{attribute 'linkalways'} 
{attribute 'no_explicit_call' := 'This FB is a CLASS and must be accessed using methods or properties'}
{attribute 'enable_dynamic_creation'}
FUNCTION_BLOCK Node_F_VN_MedianElementElementwise_UDINT EXTENDS VisionNode
VAR
    ipContainer : _ITcVnContainer;
    nMedian : _UDINT(0);
    hrPrev : _HRESULT(S_OK);
    hresult : _HRESULT(S_OK);
END_VAR

METHOD PUBLIC  Clone : I_Node
VAR
	pNode : POINTER TO Node_F_VN_MedianElementElementwise_UDINT;
END_VAR
pNode := __NEW(Node_F_VN_MedianElementElementwise_UDINT);
Clone := pNode^;
END_METHOD

METHOD FB_init : BOOL
VAR_INPUT
	bInitRetains : BOOL; // if TRUE, the retain variables are initialized (warm start / cold start)
	bInCopyCode : BOOL;  // if TRUE, the instance afterwards gets moved into the copy code (online change)
END_VAR
AddInput('ipContainer', ipContainer);
AddInput('nMedian', nMedian);
AddInput('hrPrev', hrPrev);
AddOutput('ipContainer', ipContainer);
AddOutput('hresult',hresult);
END_METHOD

METHOD PROTECTED OnExecute : HRESULT
hresult.Value := F_VN_MedianElementElementwise_UDINT(
    ipContainer := ipContainer.Value,
    nMedian := nMedian.Value,
    hrPrev:= hrPrev.Value);
END_METHOD

METHOD PUBLIC PreExecutionCheck
VAR_INPUT
	Check : I_PreExecutionChecks;
END_VAR
Check.IsTrue(ipContainer.IsValid, 'ipContainer must be a valid container');
Check.IsTrue(ipContainer.HasType('CTcVnContainer_Vector_UDINT'), 'ipContainer contains incorrect types');
END_METHOD

END_FUNCTION_BLOCK

(* stored: Version 1.1.0.1, ProductVersion 3.1.4024.13
   POU Node_F_VN_MedianElementElementwise_UDINT: Id {d961cb50-ffab-4fa3-9d1b-28a14607034a}, SpecialFunc None
   Folder Constructor: Id {9b123a5a-203a-4634-be52-330aea14f24f}
   Method Clone: Id {3fa0f73c-6dae-4c45-88df-fe23a44b6ea2}
   Method FB_init: Id {7fcc283b-19d5-4e66-907b-61e4af2658df}
   Method OnExecute: Id {4287abd7-ffa6-4ddb-98c6-a13210dc51a8}
   Method PreExecutionCheck: Id {bc74b1de-ae0d-4b67-b72f-0696e5eff306} *)
